TYPE E_SwivelState :
(
	UNDEFINED,
    Original,
    Swiveled
)USINT;
END_TYPE

(* stored: Version 1.1.0.1, ProductVersion 3.1.4020.6
   DUT E_SwivelState: Id {2ace5178-882e-49a2-9d5e-89eb1e5747dc} *)
